FUNCTION_BLOCK FB_MqttClient
VAR_INPUT
	sTopicSub	: STRING(255);
	sTopicPub  	: STRING(255);
	sPayloadPub : STRING(255);
END_VAR
VAR_OUTPUT
END_VAR
VAR
	fbMqttClient : FB_MyMqtt;
	bSubscribed	 : BOOL;
	bSetParameter : BOOL := TRUE;
	bConnect	: BOOL := TRUE;
	bGetValue	: BOOL;
END_VAR

IF bSetParameter THEN
    bSetParameter              := FALSE;
    fbMqttClient.sHostName     := '192.168.2.103';
    fbMqttClient.nHostPort     := 1883;
//  fbMqttClient.sClientId     := 'MyTcMqttClient'; 
    fbMqttClient.sTopicPrefix  := ''; 
//  fbMqttClient.nKeepAlive    := 60; 
//  fbMqttClient.sUserName     := ;
//  fbMqttClient.sUserPassword := ; 
//  fbMqttClient.stWill        := ; 
//  fbMqttClient.stTLS         := ;
END_IF

fbMqttClient.Execute(bConnect);

IF fbMqttClient.bConnected THEN
	//Check Subscription of the Topic
	IF NOT bSubscribed THEN
		bSubscribed := fbMqttClient.Subscribe(sTopic:=sTopicSub, eQoS:=TcIotMqttQos.AtMostOnceDelivery);
	END_IF
	
	//If the payload is True, set bool value to TRUE and initiate publish
	IF fbMqttClient.sPayloadRcv = 'true' THEN
		bGetValue := TRUE;
	ELSIF fbMqttClient.sPayloadRcv = 'false' THEN
		bGetValue := FALSE;
	END_IF
	
	IF bGetValue THEN
		fbMqttClient.Publish(sTopic:= sTopicPub,pPayload:= ADR(sPayloadPub), nPayloadSize:= LEN2(ADR(sPayloadPub))+1, eQoS:= TcIotMqttQos.AtMostOnceDelivery, bRetain:= FALSE, bQueue:= FALSE );
	END_IF
END_IF

END_FUNCTION_BLOCK

(* stored: Version 1.1.0.1, ProductVersion 3.1.4024.15
   POU FB_MqttClient: Id {86a6db36-3d6c-4ae4-87ab-82cf16b80846}, SpecialFunc None *)
